{attribute 'GeneratedUsingTerminal: EK1122-0000-0018'}
{attribute addProperty BoxType "EK1122-0000-0018"}
{attribute addProperty Id "Beckhoff_ELM3xxxsub_EK1100EK1100_1FC0878B2"}
{attribute addProperty CRC "436990005"}
{attribute addProperty Size "2"}
TYPE Beckhoff_ELM3xxxEK1122_1A0BF035 EXTENDS EK1122_1FC0878B :
STRUCT
	{attribute addProperty Name "Beckhoff_ELM3xxxsub_EK1100"}
	{attribute addProperty PreviousPort "Beckhoff ELM3xxxEK1122 : D"}
	Beckhoff_ELM3xxxsub_EK1100 : EK1100_1FC0878B;
END_STRUCT
END_TYPE

(* stored: Version 1.2.0.0, ProductVersion 3.1.4024.9
   DUT Beckhoff_ELM3xxxEK1122_1A0BF035: Id {a0dbc90c-7453-48c9-b2a6-4e6824d64123} *)
